// TIA Portal V17 export
// export: Created 2025-03-05T08:01:36.9793322Z, ExportSetting WithDefaults, DisplayName Totally Integrated Automation Portal, DisplayVersion V17 Update 8, DisplayName TIA Portal Openness, DisplayVersion V17 Update 8, DisplayName TIA Portal Version Control Interface, DisplayVersion V17, DisplayName SINAMICS Startdrive Advanced, DisplayVersion V17 SP2, DisplayName SINAMICS Startdrive G110M, G120, G120C, G120D, G120P, G115D, DisplayVersion V17 SP2, DisplayName SINAMICS Startdrive G130, G150, S120, S150, SINAMICS MV, S210, DisplayVersion V17 SP2, DisplayName STEP 7 Professional, DisplayVersion V17 Update 8, DisplayName SINUMERIK ONE STEP 7 Toolbox, DisplayVersion V17 Update 12, DisplayName SINUMERIK 840D sl STEP 7 Toolbox, DisplayVersion V17 Update 12, DisplayName STEP 7 Safety, DisplayVersion V17 Update 6, DisplayName WinCC Advanced, DisplayVersion V17 Update 8
DATA_BLOCK "DB10200_PYROMETERS"   // DB10200
{ S7_Optimized_Access := 'TRUE'; DB_Accessible_From_OPC_UA := 'FALSE' }
VERSION : 0.1
// stored: AutoNumber false, DBAccessibleFromOPCUA false, DBAccessibleFromWebserver true, IsOnlyStoredInLoadMemory false, IsRetainMemResEnabled false, IsWriteProtectedInAS false, MemoryReserve 100
   VAR
      UNIT_01_PYROMETER : Struct   // UNIT 01 PYROMETER
         DEVICE_STATUS : Real;   // PYROMETER DEVICE STATUS
         PROCESS_TEMPERATURE : Real;   // PYROMETER PROCESS TEMPERATURE
         HEAD_TEMPERATURE : Real;   // PYROMETER HEAD TEMPERATURE
         T1_TEMPERATURE : Real;   // PYROMETER T1 TEMPERATURE
         T2_TEMPERATURE : Real;   // PYROMETER T2 TEMPERATURE
         CURRENT_EMISSIVITY : Real;   // PYROMETER CURRENT EMISSIVITY
         CURRENT_TRANSMISSION : Real;   // PYROMETER CURRENT TRANSMISSION
      END_STRUCT;
      UNIT_02_PYROMETER : Struct
         DEVICE_STATUS : Real;   // PYROMETER DEVICE STATUS
         PROCESS_TEMPERATURE : Real;   // PYROMETER PROCESS TEMPERATURE
         HEAD_TEMPERATURE : Real;   // PYROMETER HEAD TEMPERATURE
         T1_TEMPERATURE : Real;   // PYROMETER T1 TEMPERATURE
         T2_TEMPERATURE : Real;   // PYROMETER T2 TEMPERATURE
         CURRENT_EMISSIVITY : Real;   // PYROMETER CURRENT EMISSIVITY
         CURRENT_TRANSMISSION : Real;   // PYROMETER CURRENT TRANSMISSION
      END_STRUCT;
   END_VAR
BEGIN
END_DATA_BLOCK
